// SerialPort元件
FUNCTION_BLOCK TurboPump
VAR_INPUT
	SetTmsTemp_CmdTransId:UINT;
END_VAR
VAR_OUTPUT
	SetTmsTemp_EchoTransId : UINT;
	SetTmsTemp_ErrorCode:BYTE;
END_VAR
VAR
	
END_VAR

IF SetTmsTemp_CmdTransId <> SetTmsTemp_EchoTransId THEN
	IF SetTmsTemp_ErrorCode <> 0 THEN
		SetTmsTemp(temp:= 100);
		SetTmsTemp_ErrorCode := 1;
	END_IF
END_IF

METHOD PUBLIC SetTmsTemp
VAR_INPUT
	temp :REAL;
END_VAR
END_METHOD

END_FUNCTION_BLOCK

(* stored: Version 1.1.0.1, ProductVersion 3.1.4024.16
   POU TurboPump: Id {36053571-f0f3-40e3-af8c-80f564be8382}, SpecialFunc None
   Method SetTmsTemp: Id {b3b0f644-0087-4513-b113-740716a7842f} *)
